{attribute 'pack_mode' := '2'}
TYPE ST_HOMING :
STRUCT
  bExecute      : BIT;

  stHomingParam : ST_HomeParams;
END_STRUCT
END_TYPE

(* stored: Version 1.1.0.1, ProductVersion 3.1.4024.12
   DUT ST_HOMING: Id {5851bdcf-da46-02aa-01b5-d61c3f131726} *)
